TYPE ST_PowerMonitor_OutputField EXTENDS st_PQVoltageData:
STRUCT
	r_loadshare					: 	REAL;
	ACQuality					:	ST_PQGridQualityData;
	Powerlock					: 	ARRAY [1..3] OF ST_PQPowerData;
END_STRUCT
END_TYPE

(* stored: Version 1.1.0.1, ProductVersion 3.1.4026.18
   DUT ST_PowerMonitor_OutputField: Id {d081661a-6cb9-4458-b0a8-f5a8c188d6d3} *)
